{attribute 'qualified_only'}
VAR_GLOBAL
END_VAR

(* stored: Version 1.1.0.1, ProductVersion 3.1.4024.11
   GVL Hardware_A25: Id {7f474435-78e2-4afa-9d84-b15b34687737} *)
